PROGRAM MAIN
VAR
END_VAR

Process();

END_PROGRAM

(* stored: Version 1.1.0.1, ProductVersion 3.1.4024.12
   POU MAIN: Id {6482613d-8f23-471c-bade-d42906601bb4}, SpecialFunc None *)
